FUNCTION_BLOCK EL3008
VAR
	_io : EL3xx8_Data;
	{attribute addProperty Name "WcState"}
	_wcState : WcStateInputToggle;
	{attribute addProperty Name "Info data"}
	_infoData : InfoDataAds;
END_VAR

PROPERTY IO : REFERENCE TO EL3xx8_Data
GET
IO REF= _io;
END_GET
END_PROPERTY

PROPERTY WcState : REFERENCE TO WcStateInputToggle
GET
WcState REF= _wcState;
END_GET
END_PROPERTY

END_FUNCTION_BLOCK

(* stored: Version 1.1.0.1, ProductVersion 3.1.4024.9
   POU EL3008: Id {b0321d4f-3b12-00da-3204-ce68da097e4b}, SpecialFunc None
   Property IO: Id {845e86a1-2c92-0827-06bf-cbd7eb3942d0}
   Get Get: Id {285c7a04-5f58-0367-141c-6d1c06fe3091}
   Property WcState: Id {506f3c7a-6e00-08af-06af-716b9d036f08}
   Get Get: Id {716b08c3-cda6-0aee-3388-fae9154936bb} *)
